(* PLC project Unnamed, Unknown Unnamed 1 *)
(* stored: creationDateTime 2026-08-01T21:45:19, modificationDateTime 2026-08-01T21:45:19 *)

PROGRAM main
  VAR
    TestInput : BOOL := FALSE;
    Enable : BOOL := TRUE;
    TestOutput : BOOL := FALSE;
  END_VAR

            TestOutput := TestInput AND Enable;
          
END_PROGRAM

CONFIGURATION Config0
  RESOURCE Res0 ON PLC
    TASK MainTask(INTERVAL := T#20ms, PRIORITY := 0);
    PROGRAM MainInstance WITH MainTask : main;
  END_RESOURCE
END_CONFIGURATION
